KUKA KRL data list: dockof_3.dat

&ACCESS RVP1
&REL 128
&COMMENT PLACE GUN 3
DEFDAT  DOCKOF_3
;FOLD EXTERNAL DECLARATIONS;%{PE}%MKUKATPBASIS,%CEXT,%VCOMMON,%P
;FOLD GRIPPERTECH EXT
EXT  H50 (INT  :IN,INT  :IN,INT  :IN,GRP_TYP  :IN )
;ENDFOLD (GRIPPERTECH EXT)
;FOLD SPOTTECH EXT
EXT  USERSPOT (S_COMMAND  :IN,SPOT_TYPE  :IN )
;ENDFOLD (SPOTTECH EXT)
;FOLD BASISTECH EXT;%{PE}%MKUKATPBASIS,%CEXT,%VEXT,%P
EXT  BAS (BAS_COMMAND  :IN,REAL  :IN )
DECL INT SUCCESS
;ENDFOLD (BASISTECH EXT)
;FOLD USER EXT;%{E}%MKUKATPUSER,%CEXT,%VEXT,%P
;Make here your modifications
;ENDFOLD (USER EXT)
;ENDFOLD (EXTERNAL DECLERATIONS)
;*      FDAT Declarations     *

;******************************
;*     E6POS Declarations     *
;******************************

DECL E6POS XP10={X -889.436584,Y 2792.34692,Z 1049.42603,A -106.690697,B 85.8011322,C -106.605904,S 2,T 11,E1 -1703.68701,E2 0.0,E3 0.0,E4 0.0,E5 0.0,E6 0.0}
DECL E6POS XP20={X -1220.47095,Y 2792.36401,Z 1049.43799,A -106.694199,B 85.8019104,C -106.609497,S 2,T 11,E1 -1703.68298,E2 0.0,E3 0.0,E4 0.0,E5 0.0,E6 0.0}
DECL E6POS XP30={X -1167.96106,Y 3118.54199,Z -74.9048996,A -17.4837303,B 75.0385284,C -13.4647598,S 2,T 11,E1 -1685.16003,E2 0.0,E3 0.0,E4 0.0,E5 0.0,E6 0.0}
DECL E6POS XP40={X -1175.68604,Y 3102.85791,Z -557.237915,A -13.93503,B 72.9760132,C -12.5831003,S 2,T 3,E1 -1700.55298,E2 0.0,E3 0.0,E4 0.0,E5 0.0,E6 0.0}
DECL E6POS XP50={X -1220.49194,Y 3106.99609,Z -698.499512,A -13.5889196,B 72.6338501,C -12.8622303,S 2,T 3,E1 -1703.68298,E2 0.0,E3 0.0,E4 0.0,E5 0.0,E6 0.0}
DECL E6POS XP60={X -1220.49194,Y 3106.98706,Z -746.668518,A -13.5897799,B 72.633667,C -12.8625603,S 2,T 3,E1 -1703.68103,E2 0.0,E3 0.0,E4 0.0,E5 0.0,E6 0.0}
DECL E6POS XP70={X -1433.28601,Y 3103.76392,Z 492.336212,A 58.8653717,B -0.296676606,C -179.599503,S 2,T 3,E1 -1703.68298,E2 0.0,E3 0.0,E4 0.0,E5 0.0,E6 0.0}
DECL E6POS XP80={X -1438.203,Y 3108.66406,Z 602.021484,A 58.8644714,B -0.305143893,C -179.601196,S 2,T 3,E1 -1703.68298,E2 0.0,E3 0.0,E4 0.0,E5 0.0,E6 0.0}
DECL E6POS XP90={X -856.519775,Y 3101.86792,Z 1602.84705,A 0.0745712072,B 25.8536091,C -137.305893,S 6,T 27,E1 -1428.66797,E2 0.0,E3 0.0,E4 0.0,E5 0.0,E6 0.0}

;******************************
;*     FDAT Declarations      *
;******************************

DECL FDAT FP10={TOOL_NO 3,BASE_NO 0,IPO_FRAME #BASE}
DECL FDAT FP20={TOOL_NO 3,BASE_NO 0,IPO_FRAME #BASE}
DECL FDAT FP30={TOOL_NO 3,BASE_NO 0,IPO_FRAME #BASE}
DECL FDAT FP40={TOOL_NO 3,BASE_NO 0,IPO_FRAME #BASE}
DECL FDAT FP50={TOOL_NO 3,BASE_NO 0,IPO_FRAME #BASE}
DECL FDAT FP60={TOOL_NO 3,BASE_NO 0,IPO_FRAME #BASE}
DECL FDAT FP70={TOOL_NO 10,BASE_NO 0,IPO_FRAME #BASE}
DECL FDAT FP80={TOOL_NO 10,BASE_NO 0,IPO_FRAME #BASE}
DECL FDAT FP90={TOOL_NO 10,BASE_NO 0,IPO_FRAME #BASE}

;******************************
;*  PDAT & LDAT Declarations  *
;******************************

DECL PDAT PH={VEL 100.0,ACC 100.0,APO_DIST 100.0}
DECL LDAT LH={VEL 2.0,ACC 100.0,APO_DIST 100.0,APO_FAC 50.0,ORI_TYP #VAR}

DECL E6POS XP100={X -268.887787,Y 1937.70703,Z 2261.6001,A 150.224701,B 20.9211407,C 81.1930923,S 6,T 59,E1 -735.491699,E2 0.0,E3 0.0,E4 0.0,E5 0.0,E6 0.0}
DECL FDAT FP100={TOOL_NO 10,BASE_NO 0,IPO_FRAME #BASE,POINT2[] " "}
ENDDAT
